// TwinCAT 3 PLC project PlcIotMqttSampleGoogleIoT
// ProgramVersion: 3.1.4022.4
// libraries:
//   Tc2_Standard, * (Beckhoff Automation GmbH)
//   Tc2_System, * (Beckhoff Automation GmbH)
//   Tc2_Utilities, * (Beckhoff Automation GmbH)
//   Tc3_IotBase, * (Beckhoff Automation GmbH)
//   Tc3_JsonXml, * (Beckhoff Automation GmbH)
//   Tc3_Module, * (Beckhoff Automation GmbH)
// project tree:
//   / PlcTask.TcTTO
//   POUs/ MAIN.TcPOU (not stored), PrgMqttCom.TcPOU
// real-time tasks:
//   TASK PlcTask: cycle T#10ms, priority 20, ADS port 350

CONFIGURATION PlcIotMqttSampleGoogleIoT
    RESOURCE PLC ON TwinCAT3
        TASK PlcTask(INTERVAL := T#10ms, PRIORITY := 20);
        PROGRAM MAIN WITH PlcTask : MAIN;
    END_RESOURCE
END_CONFIGURATION

// ---- POUs/PrgMqttCom.TcPOU
PROGRAM PrgMqttCom
VAR
	(* MQTT function block *)
	fbMqttClient 		: FB_IotMqttClient;
	fbMessageQueue 		: FB_IotMqttMessageQueue;
	fbMessage 			: FB_IotMqttMessage;
	bSetParameter 		: BOOL := TRUE;
	bConnect 			: BOOL := TRUE;
	hrErrorOccurred 	: HRESULT;
	
	(* Application specific data for Google Iot Core connection *)
	sProjectID				: T_MaxString := 'my-projectId';	 // Iot Core defined project ID
	sRegion					: T_MaxString := 'europe-west1'; // us-central1, europe-west1, and asia-east1
	sRegistryID				: T_MaxString := 'my-registry';	 // Iot Core defined registry ID
	sDeviceID				: T_MaxString := 'my-device';	 // Iot Core defined device ID
	sFullDevicePath 		: STRING := 'projects/%s/locations/%s/registries/%s/devices/%s'; // Full device path template - Do not change !!
	sKeyFilePath			: STRING := 'C:\TwinCAT\3.1\Config\Certificates\googleIotSample\rsa_private.pem'; // device private key
	sCaFilePath				: STRING := 'c:\TwinCAT\3.1\Config\Certificates\googleIotSample\roots.pem'; // Google RootCA chain
	sTopicPubTemplate		: STRING := '/devices/%s/events'; // Publisher topic template - Do not change !!
	sTopicSubTemplate		: STRING := '/devices/%s/commands/#'; // Subscriber topic template - Do not change !!
	
	(* JWT *)
	fbJwt				: FB_JwtEncode;
	nState				: UINT;
	hResult				: HRESULT;
	sJwt				: STRING(2048); // This buffer must be big enough to hold the Jwt token contents
	sJwtPayload			: STRING(1024); // Example content: '{"aud": "my-ProjectId","iat": 1560240662,"exp": 1560327062}'
	fbJwtPayload		: FB_JsonSaxWriter;	// Used to generate the JWT
	sPrivateKeyBuffer	: STRING(2048); // This buffer must be big enough to hold the private key contents
	dtIAT 				: DT;
	dtEXP 				: DT;
	ftTemp 				: T_FileTime;
	fbGetTime 			: GETSYSTEMTIME;
	
	(* Publish *)
	sTopicPub 			: STRING(255);
  	fbJson      		: FB_JsonSaxWriter;
  	sJsonDoc    		: STRING(255);
	fbTimer 			: TON := (PT:=T#1S);
	i					: UDINT;
	j 					: REAL;
	
	(* Subscription *)
	bSubscribed 		: BOOL;
	sTopicSub 			: STRING(255);

	(* received message *)	
	{attribute 'TcEncoding':='UTF-8'}
	sTopicRcv 			: STRING(255);
	{attribute 'TcEncoding':='UTF-8'}
	sPayloadRcv 		: STRING(255);

	(* Time *)
	systime				: GETSYSTEMTIME;
	fbSystemTime    	: GETSYSTEMTIME;
	timeAsFileTime  	: T_FILETIME;
	timeAsDT        	: DT;
		
	(* Helper *)	
	fbFormatClientID 		: FB_FormatString; // Format the client id to the full device path
	fbFormatPublishTopic	: FB_FormatString;
	fbFormatSubscrTopic		: FB_FormatString;

END_VAR

CASE nState OF
	0 :
		(* Generate JWT payload *)
		sJwtPayload := GenerateJwtPayload();
		nState := 1;

	1 : 
		(* Generate JWT *)
		(* Please note that the JWT has to be refreshed periodically, which is not shown in this sample. *)
		(* https://medium.com/google-cloud/refreshing-json-web-tokens-jwts-for-google-cloud-iot-core-897318df3836 *)
		fbJwt(	bExecute:=TRUE, 
				sHeaderAlg:='RS256', 
				sPayload:=sJwtPayload,
				pKey:=ADR(sPrivateKeyBuffer),
				nKeySize:=SIZEOF(sPrivateKeyBuffer),
				sKeyFilePath:= sKeyFilePath, 
				sJwt:=sJwt, 
				nJwtSize:=SIZEOF(sJwt),
				hrErrorCode=>hResult);
		
		IF NOT fbJwt.bBusy THEN
			IF NOT fbJwt.bError THEN
				fbJwt(bExecute:=FALSE, sJwt:=sJwt);
				nState := 2;
			END_IF
		END_IF
		
	2 : 
		bSetParameter := FALSE;
		
		// Create the full device path for the MQTT client ID
		// Example path: 'projects/my-projectId/locations/europe-west1/registries/'my-registry/devices/my-device'
		fbFormatClientID(
			sFormat			:= sFullDevicePath, 
			arg1			:= f_string(sProjectID), 
			arg2			:= f_string(sRegion), 
			arg3			:= f_string(sRegistryID), 
			arg4			:= f_string(sDeviceID), 
			sOut			=> fbMqttClient.sClientId
			);
			
		fbFormatPublishTopic(
			sFormat			:= sTopicPubTemplate,
			arg1			:= f_string(sDeviceID),
			sOut			=> sTopicPub
			);
			
		fbFormatSubscrTopic(
			sFormat			:= sTopicSubTemplate,
			arg1			:= f_string(sDeviceID),
			sOut			=> sTopicSub
			);
		
		(* Broker settings for Google IoT Core *)
		fbMqttClient.sHostName:= 'mqtt.googleapis.com';
		fbMqttClient.nHostPort:= 8883;
		fbMqttClient.sUserName:= 'unused';
		fbMqttClient.sUserPassword:= sJwt; // !! Important : sUserPassword max size can be adapted via Tc3_IotBase ParameterList (cSizeOfMqttClientUserPwd)
	
		(* TLS settings for Google IoT Core connection *)
		fbMqttClient.stTLS.sCA := sCaFilePath;
		fbMqttClient.ipMessageQueue := fbMessageQueue;
		
		nState := 3;
		
	3 : 
		(* Get current system time *)
		fbSystemTime(timeLoDW =>timeAsFileTime.dwLowDateTime, timeHiDW =>timeAsFileTime.dwHighDateTime);
		timeAsDT := FILETIME_TO_DT( timeAsFileTime );
		
		fbMqttClient.Execute(bConnect);
		IF fbMqttClient.bError THEN
			// add your error logging here
			hrErrorOccurred := fbMqttClient.hrErrorCode;
		END_IF
		IF fbMessageQueue.nQueuedMessages > 0 THEN
			IF fbMessageQueue.Dequeue(fbMessage:=fbMessage) THEN
				fbMessage.GetTopic(pTopic:=ADR(sTopicRcv), nTopicSize:=SIZEOF(sTopicRcv) );
				fbMessage.GetPayload(pPayload:=ADR(sPayloadRcv), nPayloadSize:=SIZEOF(sPayloadRcv), bSetNullTermination:=FALSE);
			END_IF
		END_IF
		
		IF fbMqttClient.bConnected THEN
			IF NOT bSubscribed THEN
				bSubscribed := fbMqttClient.Subscribe(sTopic:=sTopicSub, eQoS:=TcIotMqttQos.AtMostOnceDelivery);
				IF fbMqttClient.bError THEN
					// add your error logging here
					hrErrorOccurred := fbMqttClient.hrErrorCode;
				END_IF
			END_IF
			
			(* Publish data cyclically based on Timer *)
			fbTimer(IN:=TRUE);
			IF fbTimer.Q THEN
				fbTimer(IN:=FALSE);
				(* Create some "random" data  *)
				i := i + 1;
				j := j + 0.1;
				(* Prepare JSON document *)
				fbJson.StartObject();
				fbJson.AddKey('Timestamp');
				fbJson.AddDateTime(timeAsDT);
				fbJson.AddKey('SensorData1');
				fbJson.AddReal(j);
				fbJson.AddKey('SensorData2');
				fbJson.AddDint(i);
				fbJson.EndObject();
				sJsonDoc := fbJson.GetDocument();
				fbJson.ResetDocument();
				(* Publish message *)
				fbMqttClient.Publish(	sTopic:= sTopicPub, 
										pPayload:= ADR(sJsonDoc), nPayloadSize:= LEN2(ADR(sJsonDoc)), 
										eQoS:= TcIotMqttQos.AtMostOnceDelivery, bRetain:= FALSE, bQueue:= FALSE );
				IF fbMqttClient.bError THEN
					hrErrorOccurred := fbMqttClient.hrErrorCode;
				END_IF
			END_IF
		END_IF	
		
END_CASE

METHOD GenerateJwtPayload : STRING(1024)
// Google IoT documentation for more info: https://cloud.google.com/iot/docs/how-tos/credentials/jwts
// Testing of the token can be done here: https://jwt.io/
fbGetTime(timeLoDW => ftTemp.dwLowDateTime, timeHiDW => ftTemp.dwHighDateTime);
dtIAT := FILETIME_TO_DT(ftTemp);
dtEXP := dtIAT + T#24H; // max. is 24 hours
fbJwtPayload.StartObject();
fbJwtPayload.AddKeyString('aud', sProjectID);
fbJwtPayload.AddKeyNumber('iat', DT_TO_DINT(dtIAT));
fbJwtPayload.AddKeyNumber('exp', DT_TO_DINT(dtEXP));
fbJwtPayload.EndObject();
GenerateJwtPayload := fbJwtPayload.GetDocument();
fbJwtPayload.ResetDocument();
END_METHOD

END_PROGRAM
